PROGRAM P_System
VAR
	_arrFbButton:			ARRAY[0..10] OF FB_Button;
	
	_tonInit:				TON;
END_VAR

A_System();
A_Machine();

ACTION A_Machine:

END_ACTION

ACTION A_System:
G_stSystem.stInput.bEStop:=NOT GVL.I.bEStop;
G_stSystem.stInput.bInit:=GVL.I.bStart AND GVL.I.bStop;

//GVL.Q.bBeacon_Buzzer:=G_stSystem.stOutput.bBuzzer;
GVL.Q.bRuning:=GVL.Q.bBeacon_Green:=G_stSystem.stOutput.bLightGreen;
GVL.Q.bStop:=GVL.Q.bBeacon_Red:=G_stSystem.stOutput.bLightRed;
GVL.Q.bBeacon_Yellow:=G_stSystem.stOutput.bLightYellow;




_tonInit(IN:=GVL.I.bResetAlarm , PT:=T#5S , Q=> G_stSystem.stInput.bInit , ET=> );
_arrFbButton[0](In:=G_stSystem.stInput.bStart  , CLK:=GVL.I.bStart );
_arrFbButton[1](In:=G_stSystem.stInput.bStop  , CLK:=GVL.I.bStop );
_arrFbButton[2](In:=G_stSystem.stInput.bResetAlarm  , CLK:=GVL.I.bResetAlarm );


G_stSystem.stLogConfig.bExecute:=TRUE;
G_stSystem.stLogConfig.sFilePath:='D:\PLC\Log\System';

P_Machine(StationCount:=E_Station.Length);
END_ACTION

END_PROGRAM

(* stored: Version 1.1.0.1, ProductVersion 3.1.4024.3
   POU P_System: Id {707a1596-f082-485d-a9a7-dab54eac9110}, SpecialFunc None
   Action A_Machine: Id {bad766d9-b53e-4b69-8971-767e1991fe7c}
   Action A_System: Id {ac834835-5c48-436c-baed-30b007fe8f96} *)
